{attribute 'pack_mode' := '1'}
TYPE ST_UpdateVehicleReworkDataDataIn :
STRUCT
	sCarrierID					: STRING(30);								(* Carrier ID *)
	bNOK						: BOOL;										(* Rework required *)
END_STRUCT
END_TYPE

(* stored: Version 1.1.0.1, ProductVersion 3.1.4024.5
   DUT ST_UpdateVehicleReworkDataDataIn: Id {402e3a68-a278-44c3-9993-018c28b75dfc} *)
